PROGRAM PG_Simulationshaus
VAR
	Besucher: CTU;
	RS_0: RS;
	R_TRIG_0: R_TRIG;
	R_TRIG_1: R_TRIG;
END_VAR
VAR // added by the converter: edge detectors and wires of the graphical bodies
    _w1, _w2 : BOOL;
END_VAR

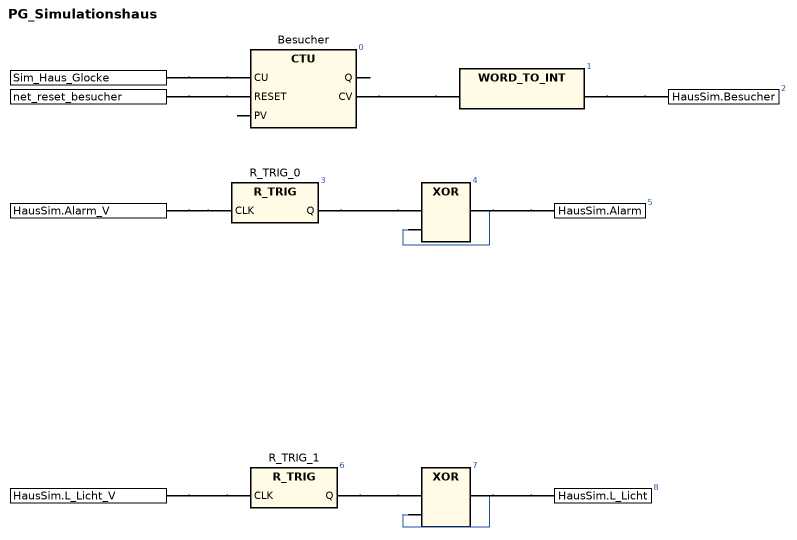
Besucher(CU := Sim_Haus_Glocke, RESET := net_reset_besucher); // CTU
HausSim.Besucher := WORD_TO_INT(Besucher.CV);
R_TRIG_0(CLK := HausSim.Alarm_V); // R_TRIG
_w1 := R_TRIG_0.Q XOR _w1;
HausSim.Alarm := _w1;
R_TRIG_1(CLK := HausSim.L_Licht_V); // R_TRIG
_w2 := R_TRIG_1.Q XOR _w2;
HausSim.L_Licht := _w2;

END_PROGRAM

(* stored: Version 1.1.0.1, ProductVersion 3.1.4018.5
   POU PG_Simulationshaus: Id {921b85e5-f626-4a34-a905-882d3266dede}, SpecialFunc None *)
